(* CoDeSys 2.3 export: ROBOT_TARGET.EXP *)

(* Data type in Robot *)
TYPE ROBOT_TARGET :
STRUCT
	Id : INT;
	MaterialIndex : INT;
	MaterialCode : BYTE;
	BoxIndex : INT;
	FirstTrack : INT;
	LastTrack : INT;
	CenterTrack : REAL;
	PickX : REAL;
	PickY : REAL;
	PickZ : REAL;
	PickAngle : REAL;
	PositionImpulses : UDINT;
	Valid : BOOL;
	InWindow : BOOL;
	Sent : BOOL;
	Picked : BOOL;
	Failed : BOOL;
	Missed : BOOL;
END_STRUCT
END_TYPE
